FUNCTION F_PosnDisp : LREAL
VAR_INPUT
	VeloInit 	: LREAL;
	VeloFinal	: LREAL;
	Accel		: LREAL;
END_VAR
VAR
END_VAR

IF Accel <> 0 THEN
	F_PosnDisp := (EXPT(VeloFinal,2) - EXPT(VeloInit,2)) / (2*Accel);
END_IF

END_FUNCTION

(* stored: Version 1.1.0.1
   POU F_PosnDisp: Id {ffc9c875-c106-052a-11df-d7882cb083dc}, SpecialFunc None *)
